// TIA Portal V15.1 export
// export: Created 2024-06-21T08:41:11.739125Z, ExportSetting WithDefaults, DisplayName Totally Integrated Automation Portal, DisplayVersion V15.1 Update 5, DisplayName TIA Portal Openness, DisplayVersion V15.1 Update 5, DisplayName SINAMICS Startdrive Advanced, DisplayVersion V15.1, DisplayName G130, G150, S120, S150, SINAMICS MV, S210, DisplayVersion V15.1, DisplayName G110M, G120, G120C, G120D, G120P, DisplayVersion V15.1, DisplayName STEP 7 Professional, DisplayVersion V15.1 Update 5, DisplayName STEP 7 Safety, DisplayVersion V15.1, DisplayName WinCC Professional, DisplayVersion V15.1 Update 5, DisplayName SIMATIC Visualization Architect, DisplayVersion V15.1
FUNCTION "LGBCalcOvertimeMoviFit" : Void   // FC6626, SCL
{ S7_Optimized_Access := 'TRUE' }
VERSION : 0.1
// stored: AutoNumber false, IsIECCheckEnabled false, SetENOAutomatically False, UDAEnableTagReadback false
   VAR_INPUT
      I_LowSpeed : Real;   // Speed value 0-100% / High speed value 0-100%
      I_HighSpeed : Real;   // Speed value 0-100% / High speed value 0-100%
      I_Diff_Pos : Real;   // Difference Positions Stop / Position Stop 1
      C_Diff_HH_LL : Real;   // Difference HH / LL
      C_ProcWarn : Real;   // Procent for Warning time
      C_ProcAlm : Real;   // Procent for Alarm time
      C_MotorRPM : Real;   // Reference RPM of the motor
      C_RatioGearbox : Real;   // Ratio Gearbox <-> Motor
      C_Diameter : Real;   // Diameter in mm
      C_Acceleration : Real;   // Acceleration in m/s²
   END_VAR
   VAR_OUTPUT
      O_RunTimeMaxWarn : DInt;   // Overtime in millisec
      O_RunTimeMaxAlm : DInt;   // Overtime in millisec
   END_VAR
   VAR_TEMP
      Diff_Pos : Real;   // Difference Positions Stop / Position Stop 1
      "m/min_HighSpeed" : Real;   // Speed in m/min
      "m/sec_HighSpeed" : Real;   // Speed in m/sec
      "m/min_LowSpeed" : Real;   // Speed in m/min
      "m/sec_LowSpeed" : Real;   // Speed in m/sec
      RampHighSpeed : Real;   // Ramp in sec
      RampLowSpeed : Real;   // Ramp in sec
      DistRampHighSpeed : Real;   // Distance Ramp in m
      DistRampLowSpeed : Real;   // Distance Ramp in m
      DistHighSpeed : Real;   // Distance High speed in m
      DistLowSpeed : Real;   // Distance Low speed in m
      TimeHighSpeed : Real;   // Time High speed in sec
      TimeLowSpeed : Real;   // Time Low speed in sec
      RunTimeMaxWarn : Real;   // Overtime in sec
      RunTimeMaxAlm : Real;   // Overtime in sec
   END_VAR
BEGIN
   // LOGIC
   IF (#I_HighSpeed <> 0.0) AND (#C_MotorRPM <> 0.0) AND (#C_RatioGearbox <> 0.0) AND (#C_Diameter <> 0.0) AND (#C_Acceleration <> 0.0) THEN
       // v = 2 * Pi * r * n [m/min] 
       #"m/min_HighSpeed" := 2 * 3.141592653 * ((#C_Diameter / 2) / 1000) * (((#I_HighSpeed / 100.0) * #C_MotorRPM) / #C_RatioGearbox);

       // v [m/sec] 
       #"m/sec_HighSpeed" := #"m/min_HighSpeed" / 60;

       // Ramp
       #RampHighSpeed := (#"m/sec_HighSpeed" / #C_Acceleration);

       // x = x0 + v0t + 1/2 * a * t² [m]
       #DistRampHighSpeed := 0 + 0 + (0.5 * #C_Acceleration * #RampHighSpeed * #RampHighSpeed);
   ELSE
       #"m/min_HighSpeed" := 0.0;
       #"m/sec_HighSpeed" := 0.0;
       #RampHighSpeed := 0.0;
       #DistRampHighSpeed := 0.0;
   END_IF;

   IF (#I_LowSpeed <> 0.0) AND (#C_MotorRPM <> 0.0) AND (#C_RatioGearbox <> 0.0) AND (#C_Diameter <> 0.0) AND (#C_Acceleration <> 0.0) THEN
       // v = 2 * Pi * r * n [m/min] 
       #"m/min_LowSpeed" := 2 * 3.141592653 * ((#C_Diameter / 2) / 1000) * (((#I_LowSpeed / 100.0) * #C_MotorRPM) / #C_RatioGearbox);

       // v [m/sec] 
       #"m/sec_LowSpeed" := #"m/min_LowSpeed" / 60;

       // Ramp
       #RampLowSpeed := (#"m/sec_LowSpeed" / #C_Acceleration);

       // x = x0 + v0t + 1/2 * a * t² [m]
       #DistRampLowSpeed := 0 + 0 + (0.5 * #C_Acceleration * #RampLowSpeed * #RampLowSpeed);
   ELSE
       #"m/min_LowSpeed" := 0.0;
       #"m/sec_LowSpeed" := 0.0;
       #RampLowSpeed := 0.0;
       #DistRampLowSpeed := 0.0;
   END_IF;

   IF (#I_Diff_Pos >= 0.0) THEN
       #Diff_Pos := #I_Diff_Pos;
   ELSE
       #Diff_Pos:= (#I_Diff_Pos * -1.0);
   END_IF;

   #DistHighSpeed := (((#Diff_Pos - #C_Diff_HH_LL) / 1000.0) - #DistRampHighSpeed);
   #TimeHighSpeed := (#DistHighSpeed / #"m/sec_HighSpeed");

   #DistLowSpeed := ((#C_Diff_HH_LL / 1000.0) - #DistRampLowSpeed);
   #TimeLowSpeed := (#DistLowSpeed / #"m/sec_LowSpeed");

   IF (#Diff_Pos <> 0.0) THEN
       #RunTimeMaxWarn := #RampHighSpeed + #TimeHighSpeed + #TimeLowSpeed + #RampLowSpeed;
       #RunTimeMaxWarn := (#RunTimeMaxWarn * (#C_ProcWarn / 100.0)) + #RunTimeMaxWarn;
       #RunTimeMaxAlm := (#RunTimeMaxWarn * (#C_ProcAlm / 100.0)) + #RunTimeMaxWarn;
   ELSE
       #RunTimeMaxWarn := 0.0;
   END_IF;

   // OUTPUT
   #O_RunTimeMaxWarn := REAL_TO_DINT(#RunTimeMaxWarn * 1000.0);
   #O_RunTimeMaxAlm := REAL_TO_DINT(#RunTimeMaxAlm * 1000.0);
END_FUNCTION
